PROGRAM P_DALI_RB3_Communication
VAR
	//INPUTS
	fbKL6821Communication		: FB_KL6821Communication;
	bResetMaximumDemandCounter	: BOOL;
	bResetOverflowCounter		: BOOL;
	bResetInactiveProcessImage	: BOOL;
	nOptions					: DWORD;
	
	//VAR_IN_OUT
	//--- See GVL_IO ---
	
	//OUTPUTS
	bBusy						: BOOL;
	bError						: BOOL;
	nErrorId					: UDINT;
	arrBufferDemandMeter		: ARRAY [0..2] OF BYTE;
	arrBufferMaximumDemandMeter	: ARRAY [0..2] OF BYTE;
	arrBufferOverflowCounter	: ARRAY [0..2] OF UINT;
	bLineIsBusy					: BOOL;
	bLineIsInitialized			: BOOL;
	bDigitalInput1Active		: BOOL;
	bDigitalInput2Active		: BOOL;
	bProcessImageInactive		: BOOL;
	bCollisionError				: BOOL;
	bPowerSupplyError			: BOOL;
	bShortCircuit				: BOOL;
END_VAR

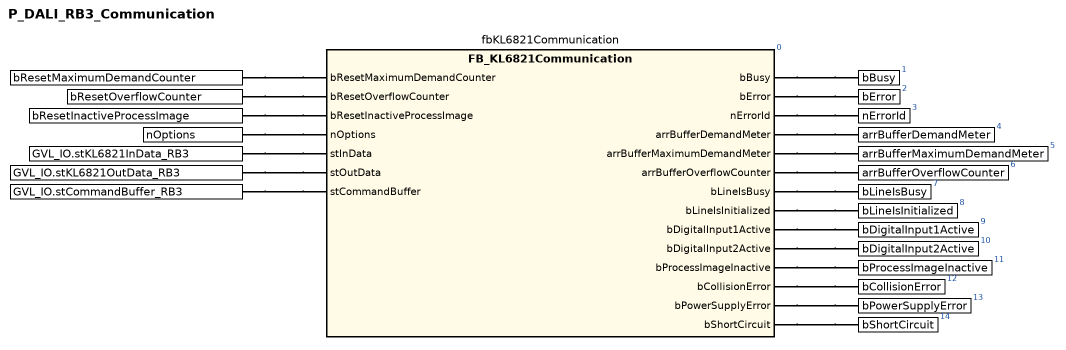
fbKL6821Communication(
    bResetMaximumDemandCounter := bResetMaximumDemandCounter,
    bResetOverflowCounter := bResetOverflowCounter,
    bResetInactiveProcessImage := bResetInactiveProcessImage,
    nOptions := nOptions,
    stInData := GVL_IO.stKL6821InData_RB3,
    stOutData := GVL_IO.stKL6821OutData_RB3,
    stCommandBuffer := GVL_IO.stCommandBuffer_RB3); // FB_KL6821Communication
bBusy := fbKL6821Communication.bBusy;
bError := fbKL6821Communication.bError;
nErrorId := fbKL6821Communication.nErrorId;
arrBufferDemandMeter := fbKL6821Communication.arrBufferDemandMeter;
arrBufferMaximumDemandMeter := fbKL6821Communication.arrBufferMaximumDemandMeter;
arrBufferOverflowCounter := fbKL6821Communication.arrBufferOverflowCounter;
bLineIsBusy := fbKL6821Communication.bLineIsBusy;
bLineIsInitialized := fbKL6821Communication.bLineIsInitialized;
bDigitalInput1Active := fbKL6821Communication.bDigitalInput1Active;
bDigitalInput2Active := fbKL6821Communication.bDigitalInput2Active;
bProcessImageInactive := fbKL6821Communication.bProcessImageInactive;
bCollisionError := fbKL6821Communication.bCollisionError;
bPowerSupplyError := fbKL6821Communication.bPowerSupplyError;
bShortCircuit := fbKL6821Communication.bShortCircuit;

END_PROGRAM

(* stored: Version 1.1.0.1, ProductVersion 3.1.4024.5
   POU P_DALI_RB3_Communication: Id {ee861f8f-0aae-465e-8399-13496db0f2fe}, SpecialFunc None *)
